{attribute 'pack_mode' := '1'}
    {attribute 'OPC.UA.DA' := '1'}
    {attribute 'OPC.UA.DA.StructuredType' := '1'}
    (*
    ST_RW_Real_Alm_Vendor_HMI_IgnitionExp
    ==================================================
    Generated from Ignition UDT: RW_Real_ALM_Vendor
    Total tags: 12
    Generated on: 2025-09-15 13:03:45
    *)
    TYPE ST_RW_Real_Alm_Vendor_HMI_IgnitionExp :
    STRUCT
        {attribute 'OPC.UA.DA' := '1'}
        Process_Alm_Val_Hi : REAL := 0.0;
        {attribute 'OPC.UA.DA' := '1'}
        Process_Alm_Val_LoLo : REAL := 0.0;
        {attribute 'OPC.UA.DA' := '1'}
        {attribute 'OPC.UA.DA.Description' := '{Description}'}
        // {Description}
        Input : REAL := 0.0;
        {attribute 'OPC.UA.DA' := '1'}
        Scale_Min : REAL := 0.0;
        {attribute 'OPC.UA.DA' := '1'}
        Process_Alm_Val_Lo : REAL := 0.0;

        {attribute 'OPC.UA.DA' := '1'}
        Process_Alm_Time_HiHi : REAL := 0.0;
        {attribute 'OPC.UA.DA' := '1'}
        Process_Alm_Time_Lo : REAL := 0.0;
        {attribute 'OPC.UA.DA' := '1'}
        Process_Alm_Time_Hi : REAL := 0.0;
        {attribute 'OPC.UA.DA' := '1'}
        HistoricalDeadband : REAL := 0.0;
        {attribute 'OPC.UA.DA' := '1'}
        Scale_Max : REAL := 0.0;

        {attribute 'OPC.UA.DA' := '1'}
        Process_Alm_Time_LoLo : REAL := 0.0;
        {attribute 'OPC.UA.DA' := '1'}
        Process_Alm_Val_HiHi : REAL := 0.0;
    END_STRUCT
    END_TYPE

(* stored: Version 1.1.0.1
   DUT ST_RW_Real_Alm_Vendor_HMI_IgnitionExp: Id {a464944d-6fdb-4ad1-a16d-adb1a261fd04} *)
